Fanuc KAREL source: kb00090.KL

-- PROVISIONAL review KL for V770-1; original PC SHA256 c0a3809f134660b1cbaaf1d109735a6d72106de9dd1e8a3fe56e0ea7b3e24d73
-- Incomplete behavior may be omitted. Consult companion uncertainty JSON. Do not deploy.
PROGRAM KB00090
%NOLOCKGROUP
BEGIN
  -- UNRESOLVED_PC offsets 5-12; opcodes 9D,23
  -- UNRESOLVED_PC offsets 17-24; opcodes 9D,23
  -- UNRESOLVED_PC offsets 29-36; opcodes 9D,23
  -- UNRESOLVED_PC offsets 41-52; opcodes 2E,23
  -- UNRESOLVED_PC offsets 57-64; opcodes 9D,23
  -- UNRESOLVED_PC offsets 69-103; opcodes 27,22,22,22,22,22,31
  -- UNRESOLVED_PC offsets 108-112; opcodes 7F
END KB00090
